//structure includes structures with TC Motion functions
TYPE ST_AxFunctions_1 :
STRUCT
	Admin				: ST_AxFunctionsAdmin_;
	PTP					: ST_AxFunctionsPTP_1;
END_STRUCT
END_TYPE

(* stored: Version 1.1.0.1, ProductVersion 3.1.4024.12
   DUT ST_AxFunctions_1: Id {be8a00d9-2abf-48be-ac44-6a555b0fbf29} *)
